FUNCTION_BLOCK Mc3Axis EXTENDS CyclicComponent IMPLEMENTS I_Initializable, I_Mc3Axis
VAR
	_Axis				 : REFERENCE TO Tc3_Mc3Ptp.AXIS_REF;
	Defaults			 : ST_Mc3MotionDefaults;
	MotionTaskCollection : Mc3MotionTaskCollection<ApplicationBaseMotionParameter.MaxMotionTasks>(THIS^);

	// Tasks
	PowerTask  : Mc3PowerTask	 := (Name := 'MC Power');
	JogTask	   : Mc3MoveJogTask	 := (Name := 'MC Jog');
	_StopTask  : I_Mc3MotionTask := Defaults.DefaultStopTask;
	_ResetTask : I_Mc3MotionTask := Defaults.DefaultResetTask;
	_HomeTask  : I_Mc3MotionTask := Defaults.DefaultHomeTask;
	SetOverride : Tc3_Mc3Ptp.MC_SetOverride;

	//
	_Initialized  : BOOL;
	_Acceleration : LREAL;
	_Deceleration : LREAL;
	_Velocity	  : LREAL;
	_Jerk		  : LREAL;
	_McBufferMode : Tc3_Mc3Ptp.EBufferMode		:= Tc3_Mc3Ptp.EBufferMode.Aborting;
	_Direction	  : Tc3_Mc3Ptp.EModuloDirection := Tc3_Mc3Ptp.EModuloDirection.ShortestDistance;
	_JogMode	  : Tc3_Mc3Ptp.EJogMode			:= Tc3_Mc3Ptp.EJogMode.StandardSlow;
END_VAR

{attribute 'monitoring' := 'call'}
PROPERTY Acceleration : LREAL
GET
Acceleration := _Acceleration;
END_GET
SET
_Acceleration := Acceleration;
END_SET
END_PROPERTY

{attribute 'monitoring' := 'call'}
PROPERTY ActualAcceleration : LREAL
GET
ActualAcceleration := _Axis.McToPlc.Act.Acceleration;
END_GET
END_PROPERTY

{attribute 'monitoring' := 'call'}
PROPERTY ActualPosition : LREAL
GET
ActualPosition := _Axis.McToPlc.Act.Position;
END_GET
END_PROPERTY

{attribute 'monitoring' := 'call'}
PROPERTY ActualPositionModulo : LREAL
GET
ActualPositionModulo := _Axis.McToPlc.Modulo.ActPosition;
END_GET
END_PROPERTY

{attribute 'monitoring' := 'call'}
PROPERTY ActualTorque : LREAL
GET
ActualTorque := _Axis.McToPlc.Act.Torque;
END_GET
END_PROPERTY

{attribute 'monitoring' := 'call'}
PROPERTY ActualVelocity : LREAL
GET
ActualVelocity := _Axis.McToPlc.Act.Velocity;
END_GET
END_PROPERTY

PROPERTY Axis : REFERENCE TO Tc3_Mc3Ptp.AXIS_REF
GET
Axis REF= _Axis;
END_GET
END_PROPERTY

PROPERTY BufferMode : REFERENCE TO Tc3_Mc3Ptp.EBufferMode
GET
BufferMode REF= _McBufferMode;
END_GET
END_PROPERTY

{attribute 'monitoring' := 'call'}
PROPERTY Busy : BOOL
GET
Busy := MotionTaskCollection.Busy;
END_GET
END_PROPERTY

METHOD CyclicLogic
IF NOT _Initialized THEN
	Initialize();
	RETURN;
END_IF

MotionTaskCollection.CyclicLogic();
END_METHOD

{attribute 'monitoring' := 'call'}
PROPERTY Coupled : BOOL
GET
Coupled := _Axis.McToPlc.Std.AxisState = EAxisState.SynchronizedMotion;
END_GET
END_PROPERTY

{attribute 'monitoring' := 'call'}
PROPERTY Deceleration : LREAL
GET
Deceleration := _Deceleration;
END_GET
SET
_Deceleration := Deceleration;
END_SET
END_PROPERTY

PROPERTY Direction : REFERENCE TO Tc3_Mc3Ptp.EModuloDirection
GET
Direction REF= _Direction;
END_GET
END_PROPERTY

{attribute 'monitoring' := 'call'}
PROPERTY Disabled : BOOL
GET
Disabled := NOT PowerTask.Enabled;
END_GET
END_PROPERTY

METHOD Disable
PowerTask.Disable();
END_METHOD

METHOD Enable
IF Error THEN
	RETURN;
END_IF

PowerTask.Enable();
END_METHOD

{attribute 'monitoring' := 'call'}
PROPERTY Enabled : BOOL
GET
Enabled := PowerTask.Enabled;
END_GET
END_PROPERTY

{attribute 'monitoring' := 'call'}
PROPERTY Error : BOOL
GET
Error := MotionTaskCollection.Error OR (_Axis.McToPlc.Std.AxisState = EAxisState.ErrorStop);
END_GET
END_PROPERTY

{attribute 'monitoring' := 'call'}
PROPERTY ErrorId : UDINT
GET
IF _Axis.McToPlc.Std.ErrorId <> 0 THEN
	ErrorId := _Axis.McToPlc.Std.ErrorId;
	RETURN;
END_IF

ErrorId := MotionTaskCollection.ErrorId;
END_GET
END_PROPERTY

(*FB_Init is always available implicitly and it is used primarily for initialization.
The return value is not evaluated. For a specific influence, you can also declare the
methods explicitly and provide additional code there with the standard initialization
code. You can evaluate the return value.*)
METHOD FB_Init : BOOL
VAR_INPUT
	(* TRUE: the retain variables are initialized (reset warm / reset cold)*)
	bInitRetains : BOOL;

	(* TRUE: the instance will be copied to the copy code afterward (online change)   *)
	bInCopyCode : BOOL;
	Name		: T_MaxString;
	Axis		: REFERENCE TO Tc3_Mc3Ptp.AXIS_REF;
END_VAR
_Axis REF= Axis;

// Register all Motion Tasks to Collection
MotionTaskCollection.AddTask(PowerTask);
MotionTaskCollection.AddTask(_StopTask);
MotionTaskCollection.AddTask(_ResetTask);
MotionTaskCollection.AddTask(_HomeTask);
MotionTaskCollection.AddTask(JogTask);
END_METHOD

METHOD Home
VAR_INPUT
END_VAR
_HomeTask.Execute();
END_METHOD

PROPERTY HomeTask : I_Mc3MotionTask
SET
MotionTaskCollection.RemoveTaskByInstance(_HomeTask);
_HomeTask := HomeTask;
MotionTaskCollection.AddTask(_HomeTask);
END_SET
END_PROPERTY

{attribute 'monitoring' := 'call'}
PROPERTY InhibitFeedBackward : BOOL
GET
InhibitFeedBackward := PowerTask.InhibitFeedBackward;
END_GET
SET
PowerTask.InhibitFeedBackward := InhibitFeedBackward;
END_SET
END_PROPERTY

{attribute 'monitoring' := 'call'}
PROPERTY InhibitFeedForward : BOOL
GET
InhibitFeedForward := PowerTask.InhibitFeedForward;
END_GET
SET
PowerTask.InhibitFeedForward := InhibitFeedForward;
END_SET
END_PROPERTY

METHOD Initialize
VAR_INST
    Sequence : UDINT;
    ReadParameter : Tc3_Mc3Ptp.MC_ReadParameter;
END_VAR
IF NOT _Initialized AND (_Axis.McToPlc.Std.AxisState <> EAxisState.Invalid) THEN
	CASE Sequence OF
		0:
			ReadParameter(Axis		  := _Axis,
						  Enable	  := TRUE,
						  ParameterId := EAxisParameterId.DefaultAcceleration,
						  Mode		  := EReadMode.Once,
						  Valid		  =>,
						  Busy		  =>,
						  Error		  =>,
						  ErrorId	  =>,
						  Value		  => _Acceleration);

			IF ReadParameter.Valid THEN
				ReadParameter(Axis := _Axis, Enable := FALSE);
				NextStep(Sequence);
			END_IF

		10:
			ReadParameter(Axis		  := _Axis,
						  Enable	  := TRUE,
						  ParameterId := EAxisParameterId.DefaultDeceleration,
						  Mode		  := EReadMode.Once,
						  Valid		  =>,
						  Busy		  =>,
						  Error		  =>,
						  ErrorId	  =>,
						  Value		  => _Deceleration);

			IF ReadParameter.Valid THEN
				ReadParameter(Axis := _Axis, Enable := FALSE);
				NextStep(Sequence);
			END_IF

		20:
			ReadParameter(Axis		  := _Axis,
						  Enable	  := TRUE,
						  ParameterId := EAxisParameterId.DefaultJerk,
						  Mode		  := EReadMode.Once,
						  Valid		  =>,
						  Busy		  =>,
						  Error		  =>,
						  ErrorId	  =>,
						  Value		  => _Jerk);

			IF ReadParameter.Valid THEN
				ReadParameter(Axis := _Axis, Enable := FALSE);
				NextStep(Sequence);
			END_IF

		30:
			ReadParameter(Axis		  := _Axis,
						  Enable	  := TRUE,
						  ParameterId := EAxisParameterId.MaximumVelocity,
						  Mode		  := EReadMode.Once,
						  Valid		  =>,
						  Busy		  =>,
						  Error		  =>,
						  ErrorId	  =>,
						  Value		  => _Velocity);

			IF ReadParameter.Valid THEN
				ReadParameter(Axis := _Axis, Enable := FALSE);
				NextStep(Sequence);
			END_IF

		40:
			Trace.LogMessage(_Name, 'Axis initialization complete');
			NextStep(Sequence);

		50:
			_Initialized := TRUE;

		999: // Error :-(
	END_CASE

	IF ReadParameter.Error AND Sequence <> 999 THEN
		Trace.LogMessage(_Name, 'Axis not initialized - error reading parameter - check links!');
		Sequence := 999;
	END_IF
END_IF
END_METHOD

{attribute 'monitoring' := 'call'}
PROPERTY Initialized : BOOL
GET
Initialized := _Initialized;
END_GET
SET
_Initialized := Initialized;
END_SET
END_PROPERTY

{attribute 'monitoring' := 'call'}
PROPERTY Jerk : LREAL
GET
Jerk := _Jerk;
END_GET
SET
_Jerk := Jerk;
END_SET
END_PROPERTY

METHOD Jog
VAR_INPUT
	JogForward	 : BOOL;
	JogBackwards : BOOL;
	Distance	 : LREAL := 0;
END_VAR
IF Error THEN
	RETURN;
END_IF

JogTask.JogBackwards := JogBackwards;
JogTask.JogForward	 := JogForward;
JogTask.Distance	 := Distance;
JogTask.Mode		 := _JogMode;
JogTask.Execute();
END_METHOD

{attribute 'monitoring' := 'call'}
PROPERTY JogMode : E_AxisJogMode
GET
IF _JogMode = Tc3_Mc3Ptp.EJogMode.StandardFast THEN
	JogMode := E_AxisJogMode.Fast;
ELSE
	JogMode := E_AxisJogMode.Slow;
END_IF
END_GET
SET
IF JogMode = E_AxisJogMode.Fast THEN
	_JogMode := Tc3_Mc3Ptp.EJogMode.StandardFast;
ELSE
	_JogMode := Tc3_Mc3Ptp.EJogMode.StandardSlow;
END_IF
END_SET
END_PROPERTY

PROPERTY MotionTasks : I_MotionTaskCollection
GET
MotionTasks := MotionTaskCollection;
END_GET
END_PROPERTY

{attribute 'monitoring' := 'call'}
PROPERTY Override : LREAL // 0-100%
SET
SetOverride(Axis		   := _Axis,
			Enable		   := TRUE,
			VelocityFactor := (Override / 100.0),
			Enabled		   =>,
			Error		   =>,
			ErrorId		   =>);
END_SET
END_PROPERTY

{attribute 'monitoring' := 'call'}
PROPERTY PositionLag : LREAL
GET
PositionLag := _Axis.McToPlc.Act.PositionLag;
END_GET
END_PROPERTY

METHOD RegisterWithParent
VAR_INPUT
	Parent : I_ContainComponents;
END_VAR
SUPER^.RegisterWithParent(Parent);
Parent.RegisterInitialize(THIS^);
END_METHOD

METHOD Reset
IF _ResetTask.Execute() THEN
	MotionTaskCollection.Reset();
END_IF
END_METHOD

PROPERTY ResetTask : I_Mc3MotionTask
SET
MotionTaskCollection.RemoveTaskByInstance(_ResetTask);
_ResetTask := ResetTask;
MotionTaskCollection.AddTask(_ResetTask);
END_SET
END_PROPERTY

{attribute 'monitoring' := 'call'}
PROPERTY SetAcceleration : LREAL
GET
SetAcceleration := _Axis.McToPlc.Set.Acceleration;
END_GET
END_PROPERTY

{attribute 'monitoring' := 'call'}
PROPERTY SetPosition : LREAL
GET
SetPosition := _Axis.McToPlc.Set.Position;
END_GET
END_PROPERTY

{attribute 'monitoring' := 'call'}
PROPERTY SetPositionModulo : LREAL
GET
SetPositionModulo := _Axis.McToPlc.Modulo.SetPosition;
END_GET
END_PROPERTY

{attribute 'monitoring' := 'call'}
PROPERTY SetVelocity : LREAL
GET
SetVelocity := _Axis.McToPlc.Set.Velocity;
END_GET
END_PROPERTY

METHOD Stop
IF Error AND _Axis.McToPlc.Std.HasError THEN
	(* It's possible that a function block errored but
	not the NC itself--in this case we can allow a stop command.
	If the NC Axis has a real fault then we want a successful reset first *)
	RETURN;
END_IF

_StopTask.Execute();
END_METHOD

{attribute 'monitoring' := 'call'}
PROPERTY Stopped : BOOL
GET
Stopped := (_Axis.McToPlc.Std.AxisState <= EAxisState.Standstill) OR ((_Axis.McToPlc.Std.AxisState = EAxisState.SynchronizedMotion) AND (SetVelocity = 0.0));
END_GET
END_PROPERTY

PROPERTY StopTask : I_Mc3MotionTask
SET
MotionTaskCollection.RemoveTaskByInstance(_StopTask);
_StopTask := StopTask;
MotionTaskCollection.AddTask(_ResetTask);
END_SET
END_PROPERTY

{attribute 'monitoring' := 'call'}
PROPERTY SynchronizedMotion : BOOL
GET
SynchronizedMotion := _Axis.McToPlc.Std.AxisState = EAxisState.SynchronizedMotion;
END_GET
END_PROPERTY

{attribute 'monitoring' := 'call'}
PROPERTY Velocity : LREAL
GET
Velocity := _Velocity;
END_GET
SET
_Velocity := Velocity;
END_SET
END_PROPERTY

END_FUNCTION_BLOCK

(* stored: Version 1.1.0.1, ProductVersion 3.1.4026.20
   POU Mc3Axis: Id {7b755d12-bde7-47e4-872e-d19b5ce399e8}, SpecialFunc None
   Folder Component: Id {322cdc66-c83d-4d9b-9af6-4b312045b224}
   Folder Cyclic: Id {4b13e22a-4196-4a05-adb9-1b8de6fccecd}
   Folder Dynamics: Id {e2766f4c-42ae-4035-911a-b08116ad2b8a}
   Folder Enable: Id {4cdfffe3-dd1a-4d83-9acb-8a813977eb21}
   Folder Home: Id {eef3d813-e6dc-43c8-b0f5-1b08f421564b}
   Folder Initialize: Id {62352c75-da34-4b3e-8f62-c1be973a80c7}
   Folder Jog: Id {c1111c46-74c9-4ed7-9895-f3e9272bb9a1}
   Folder Reset: Id {060ef385-0f6f-4a71-9be6-6e13daa0e2b0}
   Folder Settings: Id {11a9e707-af28-41b0-b73b-50567406e53e}
   Folder Status: Id {9db6bbc4-5585-49f4-9346-a377cc94d40b}
   Folder Stop: Id {aeb5218d-d539-40f1-82ca-5ac3c0a9a74b}
   Property Acceleration: Id {769983d4-87f4-42d4-8989-724adc2b60a7}
   Get Get: Id {72c60dbb-fe8b-4d09-bf78-6cb7453f610f}
   Set Set: Id {ac74071f-664b-432a-836b-9d75bd3351e9}
   Property ActualAcceleration: Id {23c7248a-c8bf-4851-b8f9-71291b83143d}
   Get Get: Id {3a174ff1-284a-479d-9ac4-07b44fb20cfb}
   Property ActualPosition: Id {19e750d4-f1cd-4c9b-bb34-2e48adf53784}
   Get Get: Id {d101b096-8c5a-4fb5-b886-817964d844e9}
   Property ActualPositionModulo: Id {9fbb5c11-401f-420c-b020-03adcd2c94a1}
   Get Get: Id {70460fff-1d82-40ed-8db5-b2e528bbc5b6}
   Property ActualTorque: Id {c43f5d3e-0ed2-4b82-bf9e-091c7cf38874}
   Get Get: Id {455ce93c-6575-40d2-9122-33f462e9a7ac}
   Property ActualVelocity: Id {3b99aa67-8ab1-42e5-9016-243f9aa2a68a}
   Get Get: Id {a495d40d-c89d-444c-a200-d292f92c3974}
   Property Axis: Id {1b536b5b-75af-4f37-9d3d-09ea16becb3f}
   Get Get: Id {92eb01af-a8cf-40dd-b37a-8435422f578e}
   Property BufferMode: Id {eb13e1b9-36ab-4361-b502-46be0db4c87f}
   Get Get: Id {3983d167-90da-4b79-8471-54cba0705403}
   Property Busy: Id {d0c93c5c-e4a6-4b4e-b0f9-a120e269ff0c}
   Get Get: Id {b0e16ae3-cf1c-4632-a624-9afcff0db000}
   Method CyclicLogic: Id {2e485cf4-3831-408a-8c77-152a2e60cb26}
   Property Coupled: Id {943bd654-d224-435a-b18b-f1fb12ee06b1}
   Get Get: Id {984a1d93-895b-4304-ba6a-c1dc47d90fdc}
   Property Deceleration: Id {3d46c410-fae9-4c59-b378-b7f0dab0d969}
   Get Get: Id {4c4b2afa-d77e-4403-a571-2cb85045e375}
   Set Set: Id {4d46e0af-a7a0-4fa3-a38d-902306c471b8}
   Property Direction: Id {6359c944-3f7f-48ff-834f-4e1a441228c7}
   Get Get: Id {95eca431-f2f6-4bdb-84b2-2369b5373842}
   Property Disabled: Id {fdde43dc-ad16-407d-9017-3887bd11b2a4}
   Get Get: Id {dd253168-820c-46ea-9e01-1735cf37f993}
   Method Disable: Id {1c391817-fa31-4646-9aa7-e76158a7ec55}
   Method Enable: Id {d365fc40-1ca8-4d17-b6b1-068ccea94484}
   Property Enabled: Id {277af7f8-31d4-4ab0-9d0b-257701ccb54c}
   Get Get: Id {c1a39a02-e71d-459d-9c26-91db453b53a1}
   Property Error: Id {63ed2f73-0c9d-4d89-a4c9-210f8ba35c0d}
   Get Get: Id {ef37721a-45c9-45ef-b64b-df7b08b0dd37}
   Property ErrorId: Id {93bf609f-fde5-49e8-8458-8115896361c9}
   Get Get: Id {8f63c5f0-46d3-4102-a8a5-b9f47d776859}
   Method FB_Init: Id {a5d95788-2be0-4ce4-a9c8-702b9ad6f90d}
   Method Home: Id {0a68f58c-2676-4c91-8b90-f5954f6894f1}
   Property HomeTask: Id {dac77fcc-8403-449c-8461-5b9445bfbef1}
   Set Set: Id {e2d829d9-c303-4f13-9b01-f9fca43f5442}
   Property InhibitFeedBackward: Id {698fde17-7a44-4025-9df6-09500bda8a2d}
   Get Get: Id {da9dfdd5-4c0f-4cfe-bafc-37d632e54688}
   Set Set: Id {55e9c50e-7070-4be9-872e-6aa8e5036779}
   Property InhibitFeedForward: Id {032b9373-0060-4019-9c6a-aa3a88e7966b}
   Get Get: Id {7d019883-5cdb-4ad1-8fa4-c6f56ee3bde4}
   Set Set: Id {893cac39-541e-48ed-8a76-92a6f129b6a9}
   Method Initialize: Id {48b8ddc2-531b-4ffa-afa5-b9951fa039dc}
   Property Initialized: Id {8378163c-34a4-41ca-b66f-85ed51788085}
   Get Get: Id {d5047218-2a28-4fa4-87fd-cd4d7d72e302}
   Set Set: Id {6668a0ab-36b3-4bd2-a45f-e98e00387112}
   Property Jerk: Id {ca39533f-d6aa-41be-8675-918ebe2fbddb}
   Get Get: Id {2c202c5a-496c-407f-9cd3-26633ce78fe6}
   Set Set: Id {ce64be9f-b543-4361-b63b-56401e4d1e0b}
   Method Jog: Id {bd10ad3a-a14e-42a8-a8e2-938896daa865}
   Property JogMode: Id {d72d3c00-19e9-4b99-881b-c351d4a98668}
   Get Get: Id {bd597374-40b6-4f74-9668-0b84e5db94e8}
   Set Set: Id {8d02dc65-41d5-43ad-9af3-df3cb9179fc5}
   Property MotionTasks: Id {8c7bb04a-df98-42d8-b950-3fc8c31ac293}
   Get Get: Id {45c069d1-a30d-4cce-b63e-950d3d777bc7}
   Property Override: Id {079ee53b-9370-4491-afb1-0b7f309a6f57}
   Set Set: Id {0ab2cf3c-ec7e-4f4a-8a18-33c61f8048b0}
   Property PositionLag: Id {8b3d61d1-c373-4f78-91fc-7b3a7f9ff790}
   Get Get: Id {e94900ad-6939-450e-9fad-6bbdf3a27e44}
   Method RegisterWithParent: Id {40d8dd85-8c4d-4f78-9eb0-0f01f278fd9e}
   Method Reset: Id {28ba2381-ae5a-4fff-ac92-decbdbee0afe}
   Property ResetTask: Id {6429039c-8bcc-4f20-8071-2f53bec22a1b}
   Set Set: Id {fb4317fc-0b94-4bc0-9403-5ae0652dfb52}
   Property SetAcceleration: Id {9b8139e6-fe0e-4210-88ee-404034908859}
   Get Get: Id {74f087f2-1f55-4492-be35-989e136f7185}
   Property SetPosition: Id {9b96b125-7e67-4dad-b5de-89800cf5fe24}
   Get Get: Id {e2536a92-71eb-4205-9d4a-0871a4986682}
   Property SetPositionModulo: Id {82f1c47e-d7aa-49d3-94a6-b3fab97dcfce}
   Get Get: Id {1383557a-d136-4b26-a7aa-e105c4b25690}
   Property SetVelocity: Id {a604cfe7-f1c8-4cde-8e44-9e828b1a9a65}
   Get Get: Id {a7210f18-ea98-49c3-ac73-7ef9ba518fe6}
   Method Stop: Id {a6e1f9e7-a7dc-4ce9-9d10-71a0c88fda01}
   Property Stopped: Id {eb504364-1142-4d8a-aeaf-e6c339ec2b03}
   Get Get: Id {61398e68-c2d5-41a6-a473-8f47af6975cd}
   Property StopTask: Id {83aabd6c-04dc-4c57-ac8f-c297822a2fe5}
   Set Set: Id {4d7620a7-cb64-423e-b169-666c783e0917}
   Property SynchronizedMotion: Id {55dfa5ef-d459-4ad6-ad57-5529fdb749d3}
   Get Get: Id {b06f9543-8987-45e3-9cc1-db3ddc240122}
   Property Velocity: Id {ee6b5cf8-e661-417f-b1b6-de5624668e88}
   Get Get: Id {fb9f768d-b4fd-4639-b7fa-f3b33e59759a}
   Set Set: Id {23174272-7941-41d8-925b-ffd67208b74b} *)
